{attribute 'qualified_only'}
VAR_GLOBAL
	AKM_Server			: STRING := 'opc.tcp://192.168.116.56:4840'; 
	FB_DCSS_Server		: STRING := 'opc.tcp://192.168.116.41:4840';
	FB_HO_Server		: STRING := 'opc.tcp://192.168.116.38:4840';
	FB_HS_Server		: STRING := 'opc.tcp://192.168.115.56:4840';
	FB_HES_Server		: STRING := 'opc.tcp://192.168.115.71:4840';
	FB_KKKW_Server		: STRING := 'opc.tcp://192.168.116.19:4840';
	FB_MV_EMAG_GT		: STRING := 'opc.tcp://192.168.116.33:4840';
	FB_MV_EMAG_VLC100	: STRING := 'opc.tcp://192.168.116.24:4840';
	FB_MV_HD			: STRING := 'opc.tcp://192.168.115.176:4840';
	FB_MV_JAVA			: STRING := 'opc.tcp://192.168.116.48:4840';
	IVA_Ofen_Read_BOOL	: STRING := 'opc.tcp://192.168.116.38:4840';
	IVA_Ofen_Read_REAL	: STRING := 'opc.tcp://192.168.116.38:4840';
	PRG_Read_LREAL		: STRING := 'opc.tcp://192.168.116.38:4840';

END_VAR

(* stored: Version 1.1.0.1, ProductVersion 3.1.4024.9
   GVL Global_OPC_UA: Id {b4ed0642-4d69-4b20-8721-fe8307c6c439} *)
